// Mitsubishi GX Works2 project: 0730plc   PLC: Q02/Q02H

PROGRAM MAIN
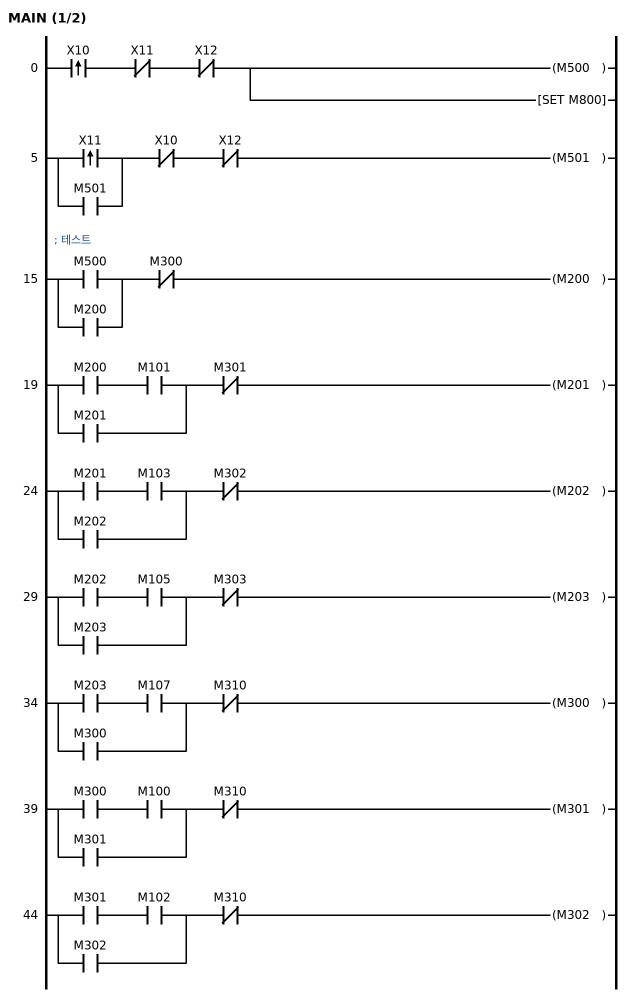
0     LDP     X10
      ANI     X11
      ANI     X12
      OUT     M500
      SET     M800
5     LDP     X11
      OR      M501
      ANI     X10
      ANI     X12
      OUT     M501
; 테스트
15    LD      M500
      OR      M200
      ANI     M300
      OUT     M200
19    LD      M200
      AND     M101
      OR      M201
      ANI     M301
      OUT     M201
24    LD      M201
      AND     M103
      OR      M202
      ANI     M302
      OUT     M202
29    LD      M202
      AND     M105
      OR      M203
      ANI     M303
      OUT     M203
34    LD      M203
      AND     M107
      OR      M300
      ANI     M310
      OUT     M300
39    LD      M300
      AND     M100
      OR      M301
      ANI     M310
      OUT     M301
44    LD      M301
      AND     M102
      OR      M302
      ANI     M310
      OUT     M302
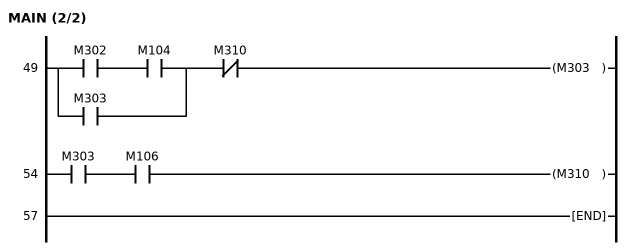
49    LD      M302
      AND     M104
      OR      M303
      ANI     M310
      OUT     M303
54    LD      M303
      AND     M106
      OUT     M310
57    END
END_PROGRAM

PROGRAM HMI
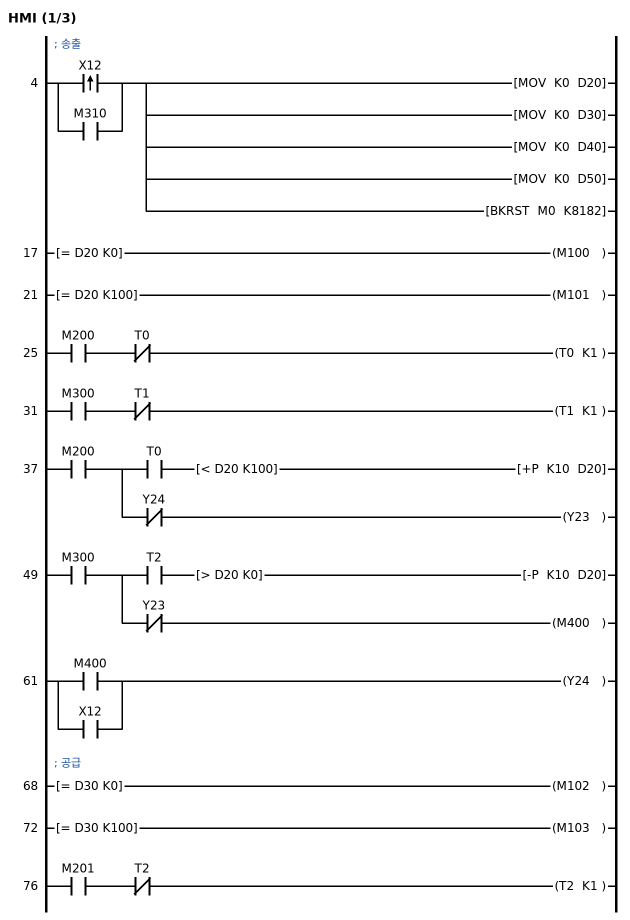
; 송출
4     LDP     X12
      OR      M310
      MOV     K0 D20
      MOV     K0 D30
      MOV     K0 D40
      MOV     K0 D50
      BKRST   M0 K8182
17    LD=     D20 K0
      OUT     M100
21    LD=     D20 K100
      OUT     M101
25    LD      M200
      ANI     T0
      OUT     T0 K1
31    LD      M300
      ANI     T1
      OUT     T1 K1
37    LD      M200
      MPS
      AND     T0
      AND<    D20 K100
      +P      K10 D20
      MPP
      ANI     Y24
      OUT     Y23
49    LD      M300
      MPS
      AND     T2
      AND>    D20 K0
      -P      K10 D20
      MPP
      ANI     Y23
      OUT     M400
61    LD      M400
      OR      X12
      OUT     Y24
; 공급
68    LD=     D30 K0
      OUT     M102
72    LD=     D30 K100
      OUT     M103
76    LD      M201
      ANI     T2
      OUT     T2 K1
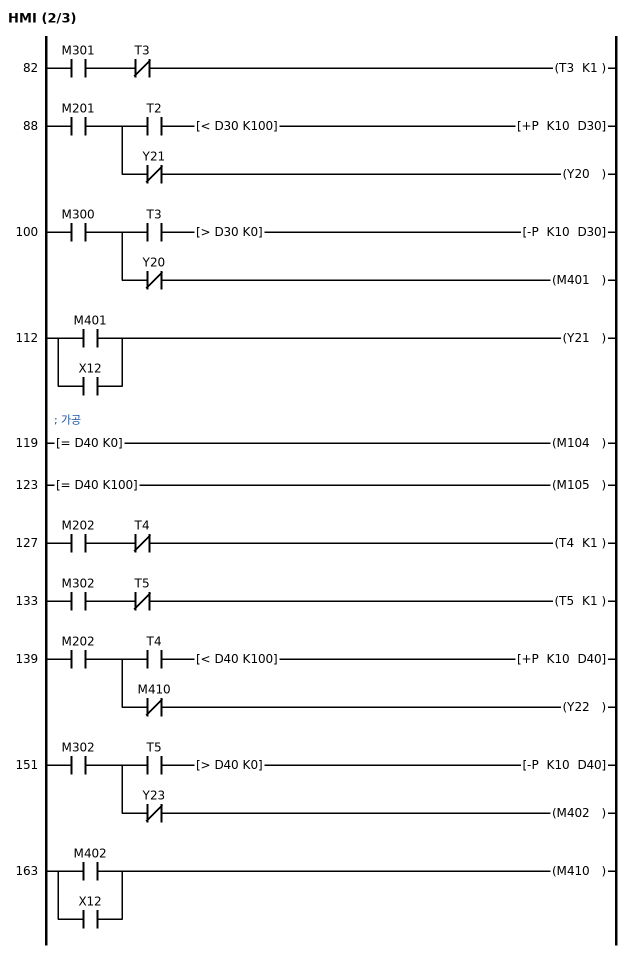
82    LD      M301
      ANI     T3
      OUT     T3 K1
88    LD      M201
      MPS
      AND     T2
      AND<    D30 K100
      +P      K10 D30
      MPP
      ANI     Y21
      OUT     Y20
100   LD      M300
      MPS
      AND     T3
      AND>    D30 K0
      -P      K10 D30
      MPP
      ANI     Y20
      OUT     M401
112   LD      M401
      OR      X12
      OUT     Y21
; 가공
119   LD=     D40 K0
      OUT     M104
123   LD=     D40 K100
      OUT     M105
127   LD      M202
      ANI     T4
      OUT     T4 K1
133   LD      M302
      ANI     T5
      OUT     T5 K1
139   LD      M202
      MPS
      AND     T4
      AND<    D40 K100
      +P      K10 D40
      MPP
      ANI     M410
      OUT     Y22
151   LD      M302
      MPS
      AND     T5
      AND>    D40 K0
      -P      K10 D40
      MPP
      ANI     Y23
      OUT     M402
163   LD      M402
      OR      X12
      OUT     M410
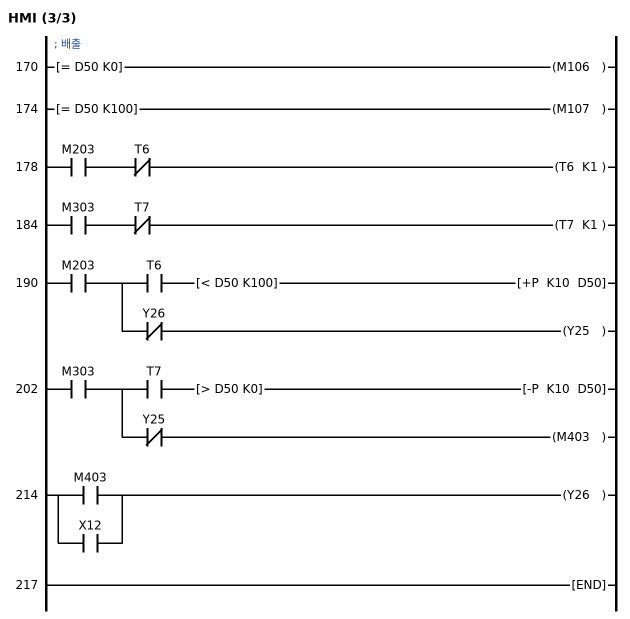
; 배출
170   LD=     D50 K0
      OUT     M106
174   LD=     D50 K100
      OUT     M107
178   LD      M203
      ANI     T6
      OUT     T6 K1
184   LD      M303
      ANI     T7
      OUT     T7 K1
190   LD      M203
      MPS
      AND     T6
      AND<    D50 K100
      +P      K10 D50
      MPP
      ANI     Y26
      OUT     Y25
202   LD      M303
      MPS
      AND     T7
      AND>    D50 K0
      -P      K10 D50
      MPP
      ANI     Y25
      OUT     M403
214   LD      M403
      OR      X12
      OUT     Y26
217   END
END_PROGRAM

PROGRAM alarm
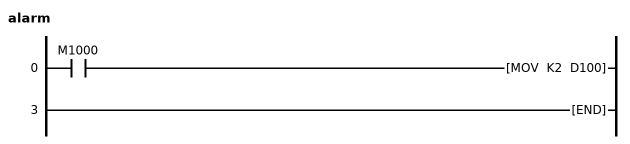
0     LD      M1000
      MOV     K2 D100
3     END
END_PROGRAM
